TYPE FW212CPolarisationFilterConfig EXTENDS DeviceConfiguration :
STRUCT
	SerialCommunication : SerialCommunication;
END_STRUCT
END_TYPE

(* stored: Version 1.1.0.1, ProductVersion 3.1.4024.4
   DUT FW212CPolarisationFilterConfig: Id {cbe37556-4961-4e39-a40e-f06d57def299} *)
